TYPE GearComRequest :
STRUCT
  Start : BOOL;
  Stop : BOOL;
  GoHome : BOOL;
  Halt : BOOL;
END_STRUCT
END_TYPE

(* stored: Version 1.1.0.1
   DUT GearComRequest: Id {9a807700-acdf-404f-9270-fa4af62f1fe6} *)
